(* IEC 61131-3 sources: teller/JD_Teller_LC2_V11/Class/Signal_Splitter_BG_Teller, 1 file *)

(* ---- Signal_Splitter_BG_Teller.st ---- *)
(*!
<Class
	Name               = "Signal_Splitter_BG_Teller"
	Revision           = "1.0"
	RealtimeTask       = "false"
	CyclicTask         = "false"
	BackgroundTask     = "true"
	DefBackground      = "100 ms"
	Sigmatek           = "false"
	OSInterface        = "false"
	HighPriority       = "false"
	Automatic          = "false"
	UpdateMode         = "Prescan"
	SharedCommandTable = "true"
	Objectsize         = "(540,120)">
	<Channels>
		<Server Name="ClassSvr" Visualized="false" Initialize="false" WriteProtected="true" Retentive="false"/>
		<Server Name="WriteValue" Visualized="true" Initialize="false" WriteProtected="false" Retentive="false"/>
		<Client Name="c_WriteValue01" Required="false" Internal="false"/>
	</Channels>
	<RevDoku>
		<Owner Company="JD" Author="SV"/>
		<Dokumentation Revision="0.0" Date="2014-09-04" Author="SV" Company="JD" Description="Kopie van Signal_Splitter_BG ref 0.0. Aangepast tot 1 client."/>
	</RevDoku>
</Class>
*)
Signal_Splitter_BG_Teller : CLASS
  //Servers:
	ClassSvr 	: SvrChCmd_DINT;
	WriteValue 	: SvrCh_DINT;
  //Clients:
	c_WriteValue01 	: CltCh_DINT;
  //Variables:
  //Functions:

	FUNCTION VIRTUAL GLOBAL Background
		VAR_INPUT
			EAX 	: UDINT;
		END_VAR
		VAR_OUTPUT
			state (EAX) 	: UDINT;
		END_VAR;

	FUNCTION VIRTUAL GLOBAL WriteValue::Write
		VAR_INPUT
			input (EAX) 	: DINT;
		END_VAR
		VAR_OUTPUT
			result (EAX) 	: DINT;
		END_VAR;
  //Tables:
	FUNCTION @STD
		VAR_OUTPUT
			ret_code	: CONFSTATES;
		END_VAR;
	FUNCTION GLOBAL TAB @CT_;
END_CLASS;

FUNCTION VIRTUAL GLOBAL Signal_Splitter_BG_Teller::WriteValue::Write
	VAR_INPUT
		input (EAX) 	: DINT;
	END_VAR
	VAR_OUTPUT
		result (EAX) 	: DINT;
	END_VAR

	WriteValue := input;

  c_WriteValue01.Write (WriteValue);

	result := WriteValue;

END_FUNCTION

FUNCTION VIRTUAL GLOBAL Signal_Splitter_BG_Teller::Background
	VAR_INPUT
		EAX 	: UDINT;
	END_VAR
	VAR_OUTPUT
		state (EAX) 	: UDINT;
	END_VAR

  WriteValue := c_WriteValue01.Read();

	state := READY;

END_FUNCTION
